// TIA Portal V20 export
// export: Created 2026-07-10T11:12:33.6709798Z, ExportSetting WithDefaults, DisplayName Totally Integrated Automation Portal, DisplayVersion V20, DisplayName TIA Portal Openness, DisplayVersion V20, DisplayName TIA Portal Version Control Interface, DisplayVersion V20, DisplayName STEP 7 Professional, DisplayVersion V20, DisplayName STEP 7 Safety, DisplayVersion V20, DisplayName WinCC Basic/Comfort/Advanced, DisplayVersion V20, DisplayName WinCC Unified, DisplayVersion V20
FUNCTION_BLOCK "MotorAdjustmentNoFeedback"   // FB14, SCL
{ S7_Optimized_Access := 'TRUE' }
VERSION : 0.1
// stored: AutoNumber true, IsIECCheckEnabled false, IsRetainMemResEnabled false, MemoryReserve 100, SetENOAutomatically false, UDAEnableTagReadback false
   VAR_INPUT
      Enable : Bool;
      Start : Bool;
      Cancel : Bool;
      AbortTime : Time := T#120s;
      MovePause : Time := T#10s;
      isMoving : Bool;
      LimitSwitch0 : Bool;
      LimitSwitch100 : Bool;
   END_VAR
   VAR_OUTPUT
      Busy : Bool;
      Error : Bool;
      Open : Bool;
      Close : Bool;
   END_VAR
   VAR_IN_OUT
      Done : Word;
      FullMovingTime : Real;
   END_VAR
   VAR
      "step" : Word;
      StartRTrig { S7_SetPoint := 'True'} : R_TRIG;
      CancelRTrig { S7_SetPoint := 'True'} : R_TRIG;
      MovingTOF { S7_SetPoint := 'True'} : TOF_TIME;
      MovingTON { S7_SetPoint := 'True'} : TON_TIME;
      PauseTON { S7_SetPoint := 'True'} : TON_TIME;
   END_VAR
BEGIN
   #StartRTrig(CLK:=#Start);
   IF #StartRTrig.Q AND #step = 0 THEN
       #step := 1;
   END_IF;

   #CancelRTrig(CLK:=#Cancel);

   IF #CancelRTrig.Q THEN
       #step := 0;
       #Error := FALSE;
   END_IF;

   IF NOT #Enable THEN
       #step := 0;
   END_IF;

   #MovingTOF(IN:=#isMoving,
              PT:=#MovePause);


   CASE #step OF
       1:
           #Busy := TRUE;
           #Done := 0;
           #Error := FALSE;
           IF NOT #MovingTOF.Q THEN
               #step += 1;
           END_IF;

       2:
           #Open := FALSE;
           #Close := TRUE;
           #step += 1;
       3:
           #MovingTON(IN := TRUE,
                      PT := #AbortTime);
           IF #LimitSwitch0 THEN
               #step += 1;
               RESET_TIMER(#MovingTON);
           END_IF;
           IF #MovingTON.Q THEN
               #Error := TRUE;
               RESET_TIMER(#MovingTON);
               #step := 10;
           END_IF;
       4:
           #Open := FALSE;
           #Close := FALSE;
           #PauseTON(IN := TRUE,
                     PT := #MovePause);
           IF #PauseTON.Q THEN
               RESET_TIMER(#PauseTON);
               #step += 1;
           END_IF;
       5:
           #Open := True;
           #Close := FALSE;
           #step += 1;
       6:
           #MovingTON(IN := TRUE,
                      PT := #AbortTime);
           #step += 1;
       7:
           IF #LimitSwitch100 THEN
               #step += 1;
           END_IF;
           IF #MovingTON.Q THEN
               #Error := True;
               RESET_TIMER(#MovingTON);
               #step := 10;
           END_IF;
       8:
           #FullMovingTime := DINT_TO_REAL(IN := #MovingTON.ET) / 1000;
           RESET_TIMER(#MovingTON);
           #step += 1;
       9:
           #Open := FALSE;
           #Close := FALSE;
           #PauseTON(IN := TRUE,
                     PT := #MovePause);
           IF #PauseTON.Q THEN
               #step += 1;
           END_IF;
       10:
           #Busy := FALSE;
           #Done := BOOL_TO_WORD(NOT #Error);
           #step := 0;  
       ELSE
           #step := 0;
           #Open := FALSE;
           #Close := FALSE;
           #Busy := FALSE;
           RESET_TIMER(#MovingTON);
           RESET_TIMER(#PauseTON);
   END_CASE;
END_FUNCTION_BLOCK
